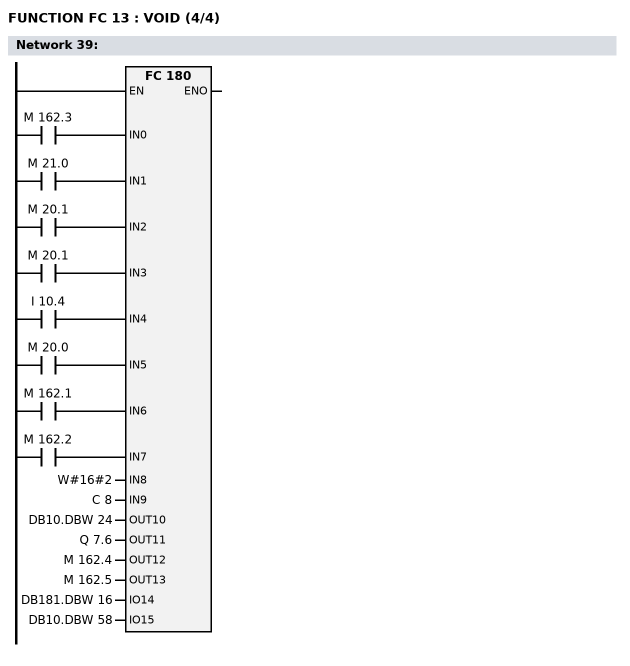

      A     M    162.3;
      =     L      4.0;
      BLD   103;
      A     M     21.0;
      =     L      4.1;
      BLD   103;
      A     M     20.1;
      =     L      4.2;
      BLD   103;
      A     M     20.1;
      =     L      4.3;
      BLD   103;
      A     I     10.4;
      =     L      4.4;
      BLD   103;
      A     M     20.0;
      =     L      4.5;
      BLD   103;
      A     M    162.1;
      =     L      4.6;
      BLD   103;
      A     M    162.2;
      =     L      4.7;
      BLD   103;
      CALL FC   180 (
           IN0                      := L      4.0,
           IN1                      := L      4.1,
           IN2                      := L      4.2,
           IN3                      := L      4.3,
           IN4                      := L      4.4,
           IN5                      := L      4.5,
           IN6                      := L      4.6,
           IN7                      := L      4.7,
           IN8                      := W#16#2,
           IN9                      := C      8,
           OUT10                    := DB10.DBW   24,
           OUT11                    := Q      7.6,
           OUT12                    := M    162.4,
           OUT13                    := M    162.5,
           IO14                     := DB181.DBW   16,
           IO15                     := DB10.DBW   58);
      NOP   0;
END_FUNCTION

FUNCTION FC 14 : VOID
TITLE =
AUTHOR : Xaadem <yalanci63@yahoo.com>
FAMILY : DRIVES
NAME : DRIVES
VERSION : 0.1


VAR_TEMP
  TEMP0 : REAL ;
END_VAR
BEGIN
NETWORK
TITLE =
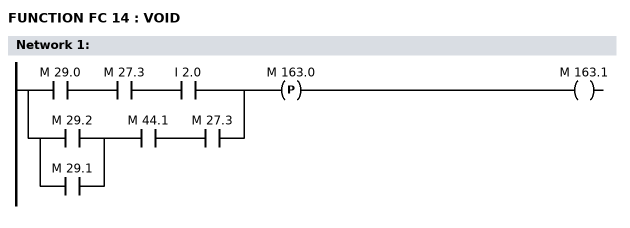

      A(    ;
      A     M     29.0;
      A     M     27.3;
      A     I      2.0;
      O     ;
      A(    ;
      O     M     29.2;
      O     M     29.1;
      )     ;
      A     M     44.1;
      A     M     27.3;
      )     ;
      FP    M    163.0;
      =     M    163.1;
NETWORK
TITLE =

      A     M     29.0;
      AN    I      2.1;
      O     ;
      A(    ;
      O     M     29.2;
      O     M     29.1;
      )     ;
      AN    M     44.1;
      A(    ;
      AN    T     25;
      L     DB2.DBW   58;
      SD    T     29;
      NOP   0;
      NOP   0;
      NOP   0;
      A     T     29;
      )     ;
      O     M     11.1;
      =     M    163.2;
NETWORK
TITLE =

      AN    M    179.0;
      AN    M    180.0;
      AN    M    181.0;
      AN    M    182.0;
      AN    M    183.0;
      A(    ;
      O     I      1.6;
      O     I      4.2;
      )     ;
      A(    ;
      A(    ;
      A     I     10.5;
      L     DB2.DBW   60;
      SD    T     30;
      NOP   0;
      NOP   0;
      NOP   0;
      A     T     30;
      )     ;
      AN    M    155.7;
      NOT   ;
      )     ;
      AN    M    206.0;
      AN    M    207.0;
      =     M    163.3;
NETWORK
TITLE =
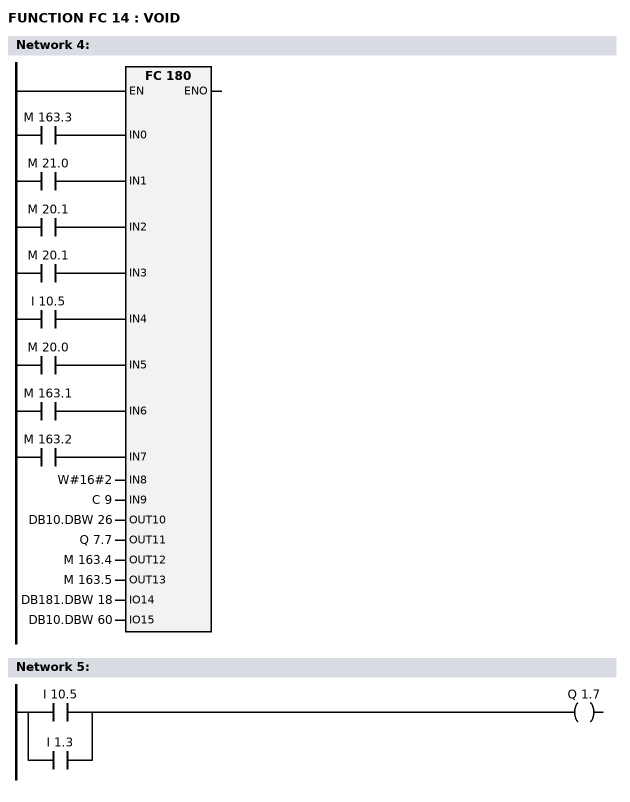

      A     M    163.3;
      =     L      4.0;
      BLD   103;
      A     M     21.0;
      =     L      4.1;
      BLD   103;
      A     M     20.1;
      =     L      4.2;
      BLD   103;
      A     M     20.1;
      =     L      4.3;
      BLD   103;
      A     I     10.5;
      =     L      4.4;
      BLD   103;
      A     M     20.0;
      =     L      4.5;
      BLD   103;
      A     M    163.1;
      =     L      4.6;
      BLD   103;
      A     M    163.2;
      =     L      4.7;
      BLD   103;
      CALL FC   180 (
           IN0                      := L      4.0,
           IN1                      := L      4.1,
           IN2                      := L      4.2,
           IN3                      := L      4.3,
           IN4                      := L      4.4,
           IN5                      := L      4.5,
           IN6                      := L      4.6,
           IN7                      := L      4.7,
           IN8                      := W#16#2,
           IN9                      := C      9,
           OUT10                    := DB10.DBW   26,
           OUT11                    := Q      7.7,
           OUT12                    := M    163.4,
           OUT13                    := M    163.5,
           IO14                     := DB181.DBW   18,
           IO15                     := DB10.DBW   60);
      NOP   0;
NETWORK
TITLE =

      O     I     10.5;
      O     I      1.3;
      =     Q      1.7;
END_FUNCTION

FUNCTION FC 15 : VOID
TITLE =
AUTHOR : Xaadem <yalanci63@yahoo.com>
FAMILY : DRIVES
NAME : DRIVES
VERSION : 0.1


VAR_TEMP
  TEMP0 : REAL ;
END_VAR
BEGIN
NETWORK
TITLE =

      A     I      0.2;
      AN    M    164.4;
      A(    ;
      A(    ;
      O     Q      0.0;
      O     I      1.0;
      O     I      2.0;
      O     I      2.4;
      O     I      2.6;
      O     I      2.7;
      O(    ;
      A     I      4.1;
      FP    M    209.2;
      )     ;
      )     ;
      =     M    209.3;
      A     M    209.3;
      )     ;
      FP    M    164.0;
      =     M    164.1;
NETWORK
TITLE =

      A(    ;
      A     M     38.0;
      A(    ;
      O     I     11.4;
      O     I     12.5;
      )     ;
      L     DB2.DBW   62;
      SD    T     31;
      NOP   0;
      NOP   0;
      NOP   0;
      A     T     31;
      )     ;
      FP    M    209.0;
      =     M    164.2;
NETWORK
TITLE =
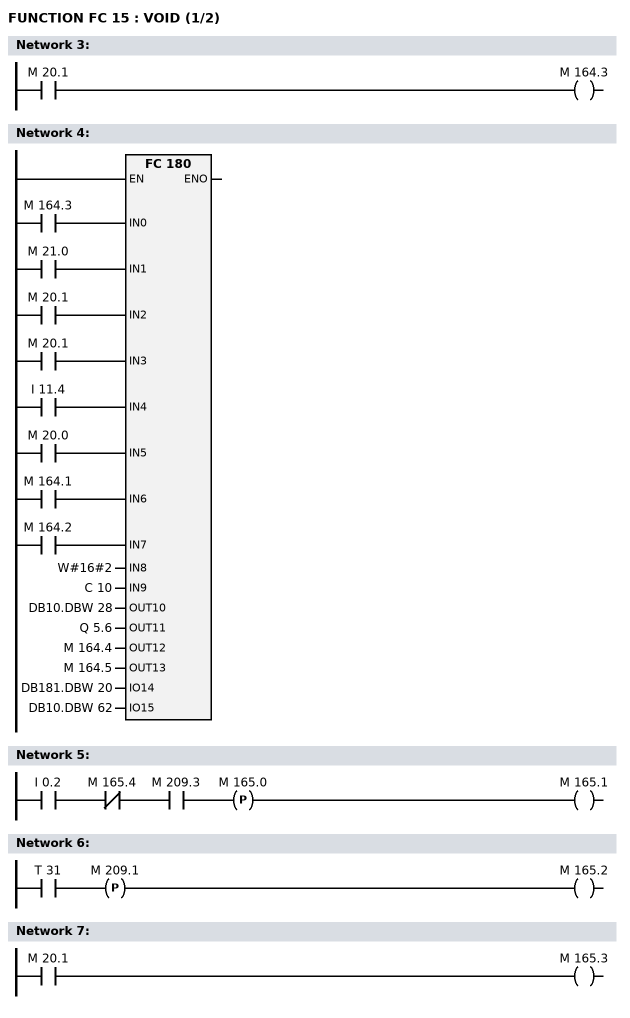

      A     M     20.1;
      =     M    164.3;
NETWORK
TITLE =

      A     M    164.3;
      =     L      4.0;
      BLD   103;
      A     M     21.0;
      =     L      4.1;
      BLD   103;
      A     M     20.1;
      =     L      4.2;
      BLD   103;
      A     M     20.1;
      =     L      4.3;
      BLD   103;
      A     I     11.4;
      =     L      4.4;
      BLD   103;
      A     M     20.0;
      =     L      4.5;
      BLD   103;
      A     M    164.1;
      =     L      4.6;
      BLD   103;
      A     M    164.2;
      =     L      4.7;
      BLD   103;
      CALL FC   180 (
           IN0                      := L      4.0,
           IN1                      := L      4.1,
           IN2                      := L      4.2,
           IN3                      := L      4.3,
           IN4                      := L      4.4,
           IN5                      := L      4.5,
           IN6                      := L      4.6,
           IN7                      := L      4.7,
           IN8                      := W#16#2,
           IN9                      := C     10,
           OUT10                    := DB10.DBW   28,
           OUT11                    := Q      5.6,
           OUT12                    := M    164.4,
           OUT13                    := M    164.5,
           IO14                     := DB181.DBW   20,
           IO15                     := DB10.DBW   62);
      NOP   0;
NETWORK
TITLE =

      A     I      0.2;
      AN    M    165.4;
      A     M    209.3;
      FP    M    165.0;
      =     M    165.1;
NETWORK
TITLE =

      A     T     31;
      FP    M    209.1;
      =     M    165.2;
NETWORK
TITLE =

      A     M     20.1;
      =     M    165.3;
NETWORK
TITLE =
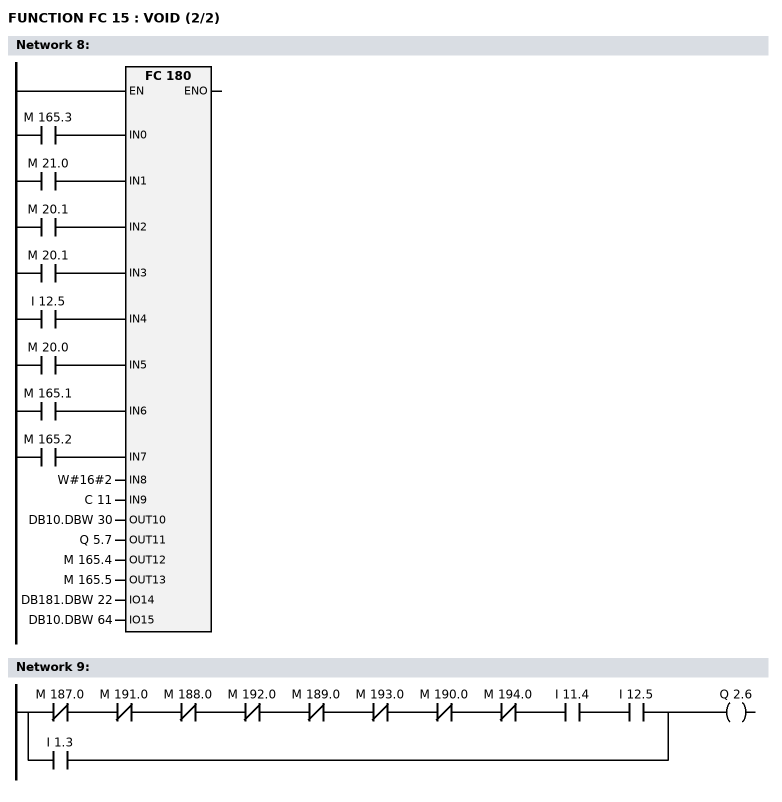

      A     M    165.3;
      =     L      4.0;
      BLD   103;
      A     M     21.0;
      =     L      4.1;
      BLD   103;
      A     M     20.1;
      =     L      4.2;
      BLD   103;
      A     M     20.1;
      =     L      4.3;
      BLD   103;
      A     I     12.5;
      =     L      4.4;
      BLD   103;
      A     M     20.0;
      =     L      4.5;
      BLD   103;
      A     M    165.1;
      =     L      4.6;
      BLD   103;
      A     M    165.2;
      =     L      4.7;
      BLD   103;
      CALL FC   180 (
           IN0                      := L      4.0,
           IN1                      := L      4.1,
           IN2                      := L      4.2,
           IN3                      := L      4.3,
           IN4                      := L      4.4,
           IN5                      := L      4.5,
           IN6                      := L      4.6,
           IN7                      := L      4.7,
           IN8                      := W#16#2,
           IN9                      := C     11,
           OUT10                    := DB10.DBW   30,
           OUT11                    := Q      5.7,
           OUT12                    := M    165.4,
           OUT13                    := M    165.5,
           IO14                     := DB181.DBW   22,
           IO15                     := DB10.DBW   64);
      NOP   0;
NETWORK
TITLE =

      AN    M    187.0;
      AN    M    191.0;
      AN    M    188.0;
      AN    M    192.0;
      AN    M    189.0;
      AN    M    193.0;
      AN    M    190.0;
      AN    M    194.0;
      A     I     11.4;
      A     I     12.5;
      O     I      1.3;
      =     Q      2.6;
END_FUNCTION

FUNCTION FC 20 : VOID
TITLE =
AUTHOR : Xaadem <yalanci63@yahoo.com>
FAMILY : ANALOGUE
NAME : ANALOGUE
VERSION : 0.1


VAR_TEMP
  TEMP0 : WORD ;
  TEMP1 : REAL ;
  TEMP2 : REAL ;
END_VAR
BEGIN
NETWORK
TITLE =

      L     ID   105;
      DTR   ;
      T     #TEMP2;
      NOP   0;
NETWORK
TITLE =

      L     ID   105;
      DTR   ;
      T     DB10.DBD  264;
      NOP   0;
NETWORK
TITLE =

      A(    ;
      A     I    108.0;
      FP    M    500.0;
      L     DB2.DBW  200;
      SF    T    100;
      NOP   0;
      NOP   0;
      NOP   0;
      A     T    100;
      )     ;
      NOT   ;
      A(    ;
      A(    ;
      O     I      5.5;
      O     I      6.4;
      )     ;
      L     DB2.DBW  210;
      SD    T    105;
      NOP   0;
      NOP   0;
      NOP   0;
      A     T    105;
      )     ;
      =     M    500.1;
NETWORK
TITLE =
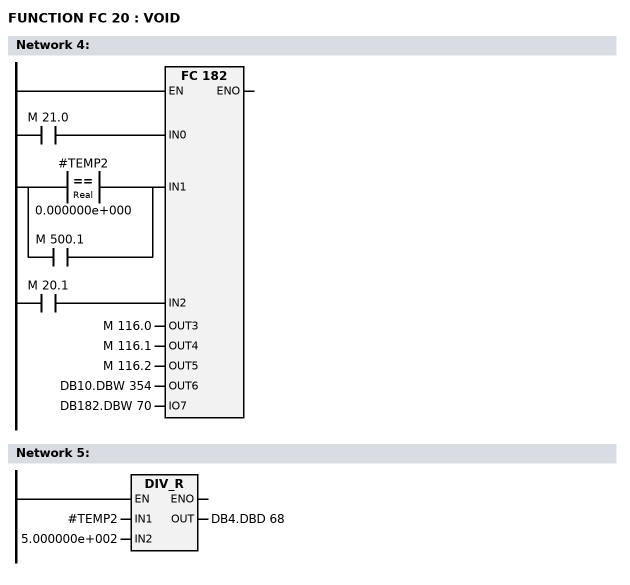

      A     M     21.0;
      =     L     10.0;
      BLD   103;
      A(    ;
      O(    ;
      L     #TEMP2;
      L     0.000000e+000;
      ==R   ;
      )     ;
      O     M    500.1;
      )     ;
      =     L     10.1;
      BLD   103;
      A     M     20.1;
      =     L     10.2;
      BLD   103;
      CALL FC   182 (
           IN0                      := L     10.0,
           IN1                      := L     10.1,
           IN2                      := L     10.2,
           OUT3                     := M    116.0,
           OUT4                     := M    116.1,
           OUT5                     := M    116.2,
           OUT6                     := DB10.DBW  354,
           IO7                      := DB182.DBW   70);
      NOP   0;
NETWORK
TITLE =

      L     #TEMP2;
      L     5.000000e+002;
      /R    ;
      T     DB4.DBD   68;
      NOP   0;
NETWORK
TITLE =

      A(    ;
      L     DB4.DBD   68;
      L     DB4.DBD   76;
      >=R   ;
      )     ;
      A(    ;
      L     DB4.DBD   68;
      L     DB4.DBD   72;
      <=R   ;
      )     ;
      =     L     10.0;
      A     L     10.0;
      BLD   102;
      =     M    172.0;
      O     L     10.0;
      O     I      1.3;
      =     Q      1.2;
      A     L     10.0;
      BLD   102;
      =     Q      3.7;
NETWORK
TITLE =

      A(    ;
      L     DB4.DBD   68;
      L     DB4.DBD   84;
      >=R   ;
      )     ;
      A(    ;
      L     DB4.DBD   68;
      L     DB4.DBD   80;
      <=R   ;
      )     ;
      =     L     10.0;
      A     L     10.0;
      BLD   102;
      =     M    172.1;
      O     L     10.0;
      O     I      1.3;
      =     Q      1.3;
      A     L     10.0;
      BLD   102;
      =     Q      4.0;
NETWORK
TITLE =
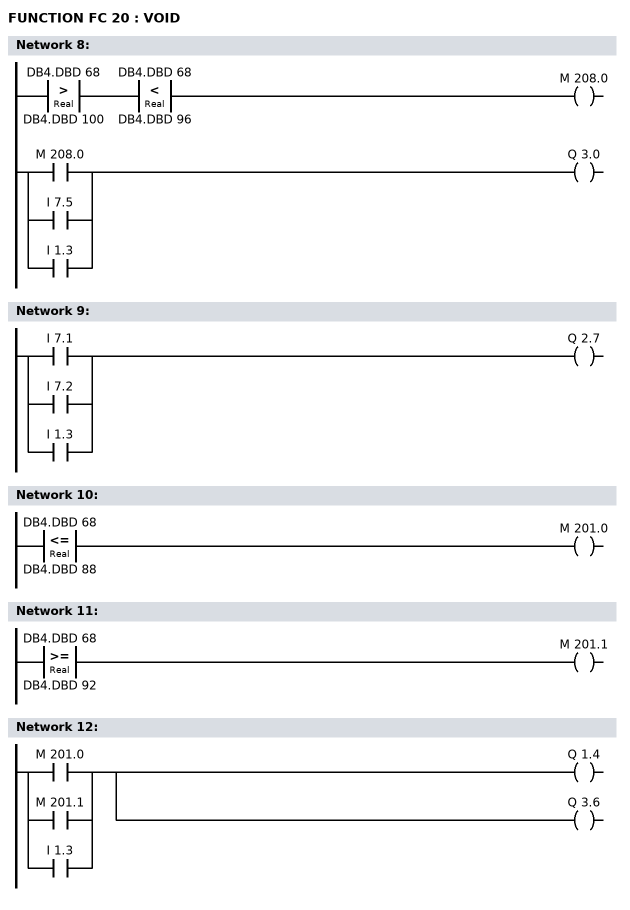

      A(    ;
      L     DB4.DBD   68;
      L     DB4.DBD  100;
      >R    ;
      )     ;
      A(    ;
      L     DB4.DBD   68;
      L     DB4.DBD   96;
      <R    ;
      )     ;
      =     M    208.0;
      A     M    208.0;
      O     I      7.5;
      O     I      1.3;
      =     Q      3.0;
NETWORK
TITLE =

      O     I      7.1;
      O     I      7.2;
      O     I      1.3;
      =     Q      2.7;
NETWORK
TITLE =

      L     DB4.DBD   68;
      L     DB4.DBD   88;
      <=R   ;
      =     M    201.0;
NETWORK
TITLE =

      L     DB4.DBD   68;
      L     DB4.DBD   92;
      >=R   ;
      =     M    201.1;
NETWORK
TITLE =

      O     M    201.0;
      O     M    201.1;
      O     I      1.3;
      =     Q      1.4;
      =     Q      3.6;
NETWORK
TITLE =

      A     M    200.6;
      A     M     20.1;
      =     L     10.0;
      A     L     10.0;
      JNB   M001;
      L     DW#16#80000000;
      T     QD   105;
M001: NOP   0;
      AN    L     10.0;
      JNB   M002;
      L     DW#16#0;
      T     QD   105;
M002: NOP   0;
NETWORK
TITLE =
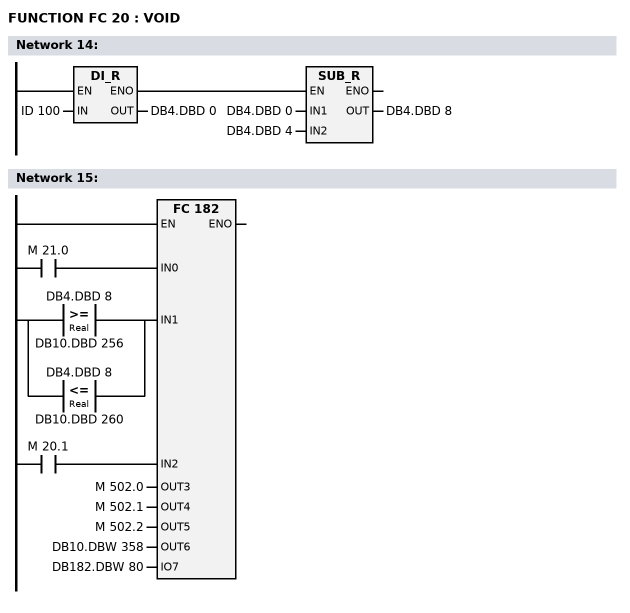

      A(    ;
      L     ID   100;
      DTR   ;
      T     DB4.DBD    0;
      SET   ;
      SAVE  ;
      CLR   ;
      A     BR;
      )     ;
      JNB   M003;
      L     DB4.DBD    0;
      L     DB4.DBD    4;
      -R    ;
      T     DB4.DBD    8;
M003: NOP   0;
NETWORK
TITLE =

      A     M     21.0;
      =     L     10.0;
      BLD   103;
      A(    ;
      O(    ;
      L     DB4.DBD    8;
      L     DB10.DBD  256;
      >=R   ;
      )     ;
      O(    ;
      L     DB4.DBD    8;
      L     DB10.DBD  260;
      <=R   ;
      )     ;
      )     ;
      =     L     10.1;
      BLD   103;
      A     M     20.1;
      =     L     10.2;
      BLD   103;
      CALL FC   182 (
           IN0                      := L     10.0,
           IN1                      := L     10.1,
           IN2                      := L     10.2,
           OUT3                     := M    502.0,
           OUT4                     := M    502.1,
           OUT5                     := M    502.2,
           OUT6                     := DB10.DBW  358,
           IO7                      := DB182.DBW   80);
      NOP   0;
NETWORK
TITLE =

      A(    ;
      L     DB4.DBD    8;
      L     DB10.DBD  248;
      >=R   ;
      )     ;
      =     M    503.1;
      A     M    503.1;
      O(    ;
      A(    ;
      L     DB4.DBD    8;
      L     DB10.DBD  252;
      <=R   ;
      )     ;
      =     M    503.2;
      A     M    503.2;
      )     ;
      =     M    503.0;
NETWORK
TITLE =

      A(    ;
      A     I    103.0;
      FP    M    501.0;
      L     DB2.DBW  202;
      SF    T    101;
      NOP   0;
      NOP   0;
      NOP   0;
      A     T    101;
      )     ;
      NOT   ;
      A     T    105;
      =     M    501.1;
NETWORK
TITLE =
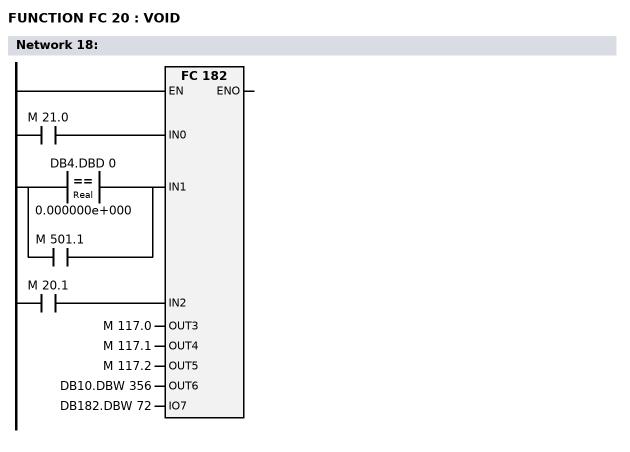

      A     M     21.0;
      =     L     10.0;
      BLD   103;
      A(    ;
      O(    ;
      L     DB4.DBD    0;
      L     0.000000e+000;
      ==R   ;
      )     ;
      O     M    501.1;
      )     ;
      =     L     10.1;
      BLD   103;
      A     M     20.1;
      =     L     10.2;
      BLD   103;
      CALL FC   182 (
           IN0                      := L     10.0,
           IN1                      := L     10.1,
           IN2                      := L     10.2,
           OUT3                     := M    117.0,
           OUT4                     := M    117.1,
           OUT5                     := M    117.2,
           OUT6                     := DB10.DBW  356,
           IO7                      := DB182.DBW   72);
      NOP   0;
NETWORK
TITLE =

      A     M     20.1;
      A     M    200.5;
      =     L     10.0;
      A     L     10.0;
      JNB   M004;
      L     DW#16#80000000;
      T     QD   100;
M004: NOP   0;
      AN    L     10.0;
      JNB   M005;
      L     DW#16#0;
      T     QD   100;
M005: NOP   0;
NETWORK
TITLE =
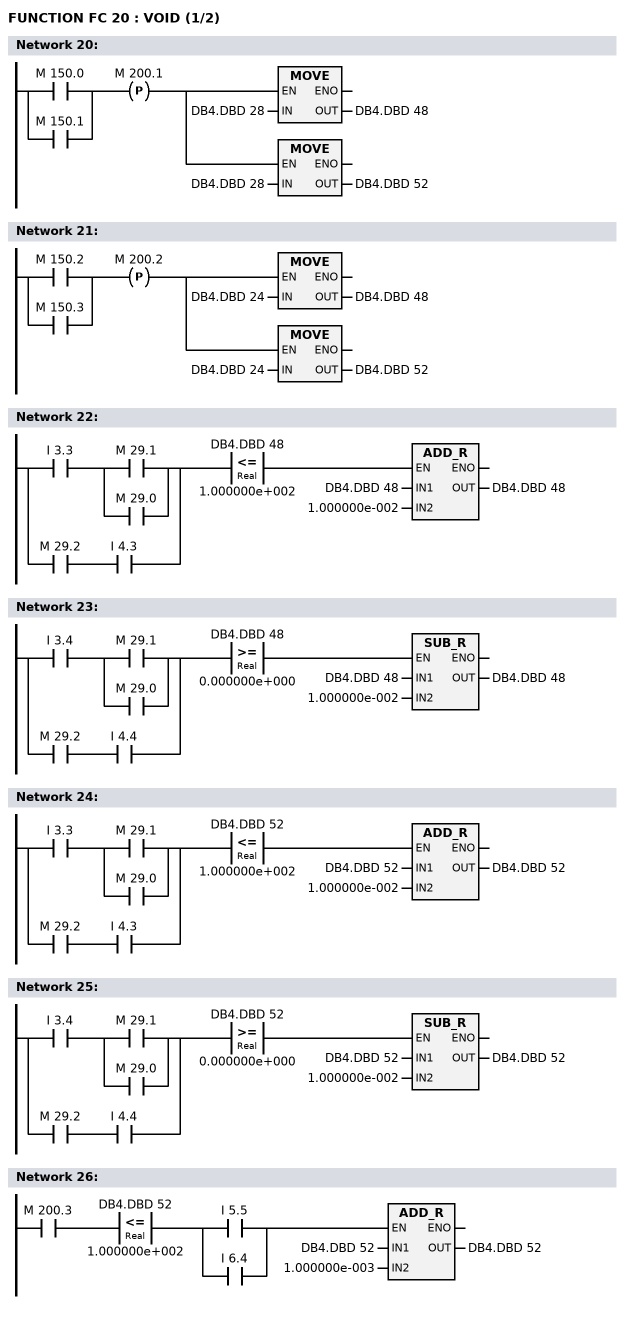

      A(    ;
      O     M    150.0;
      O     M    150.1;
      )     ;
      FP    M    200.1;
      =     L     10.0;
      A     L     10.0;
      JNB   M006;
      L     DB4.DBD   28;
      T     DB4.DBD   48;
M006: NOP   0;
      A     L     10.0;
      JNB   M007;
      L     DB4.DBD   28;
      T     DB4.DBD   52;
M007: NOP   0;
NETWORK
TITLE =

      A(    ;
      O     M    150.2;
      O     M    150.3;
      )     ;
      FP    M    200.2;
      =     L     10.0;
      A     L     10.0;
      JNB   M008;
      L     DB4.DBD   24;
      T     DB4.DBD   48;
M008: NOP   0;
      A     L     10.0;
      JNB   M009;
      L     DB4.DBD   24;
      T     DB4.DBD   52;
M009: NOP   0;
NETWORK
TITLE =

      A(    ;
      A     I      3.3;
      A(    ;
      O     M     29.1;
      O     M     29.0;
      )     ;
      O     ;
      A     M     29.2;
      A     I      4.3;
      )     ;
      A(    ;
      L     DB4.DBD   48;
      L     1.000000e+002;
      <=R   ;
      )     ;
      JNB   M00a;
      L     DB4.DBD   48;
      L     1.000000e-002;
      +R    ;
      T     DB4.DBD   48;
M00a: NOP   0;
NETWORK
TITLE =

      A(    ;
      A     I      3.4;
      A(    ;
      O     M     29.1;
      O     M     29.0;
      )     ;
      O     ;
      A     M     29.2;
      A     I      4.4;
      )     ;
      A(    ;
      L     DB4.DBD   48;
      L     0.000000e+000;
      >=R   ;
      )     ;
      JNB   M00b;
      L     DB4.DBD   48;
      L     1.000000e-002;
      -R    ;
      T     DB4.DBD   48;
M00b: NOP   0;
NETWORK
TITLE =

      A(    ;
      A     I      3.3;
      A(    ;
      O     M     29.1;
      O     M     29.0;
      )     ;
      O     ;
      A     M     29.2;
      A     I      4.3;
      )     ;
      A(    ;
      L     DB4.DBD   52;
      L     1.000000e+002;
      <=R   ;
      )     ;
      JNB   M00c;
      L     DB4.DBD   52;
      L     1.000000e-002;
      +R    ;
      T     DB4.DBD   52;
M00c: NOP   0;
NETWORK
TITLE =

      A(    ;
      A     I      3.4;
      A(    ;
      O     M     29.1;
      O     M     29.0;
      )     ;
      O     ;
      A     M     29.2;
      A     I      4.4;
      )     ;
      A(    ;
      L     DB4.DBD   52;
      L     0.000000e+000;
      >=R   ;
      )     ;
      JNB   M00d;
      L     DB4.DBD   52;
      L     1.000000e-002;
      -R    ;
      T     DB4.DBD   52;
M00d: NOP   0;
NETWORK
TITLE =

      A     M    200.3;
      A(    ;
      L     DB4.DBD   52;
      L     1.000000e+002;
      <=R   ;
      )     ;
      A(    ;
      O     I      5.5;
      O     I      6.4;
      )     ;
      JNB   M00e;
      L     DB4.DBD   52;
      L     1.000000e-003;
      +R    ;
      T     DB4.DBD   52;
M00e: NOP   0;
NETWORK
TITLE =
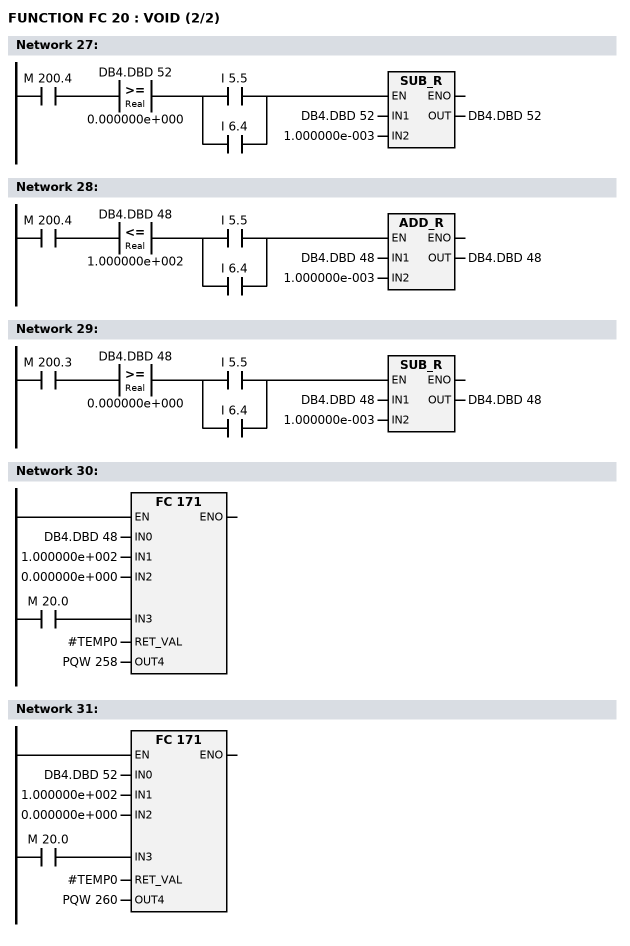

      A     M    200.4;
      A(    ;
      L     DB4.DBD   52;
      L     0.000000e+000;
      >=R   ;
      )     ;
      A(    ;
      O     I      5.5;
      O     I      6.4;
      )     ;
      JNB   M00f;
      L     DB4.DBD   52;
      L     1.000000e-003;
      -R    ;
      T     DB4.DBD   52;
M00f: NOP   0;
NETWORK
TITLE =

      A     M    200.4;
      A(    ;
      L     DB4.DBD   48;
      L     1.000000e+002;
      <=R   ;
      )     ;
      A(    ;
      O     I      5.5;
      O     I      6.4;
      )     ;
      JNB   M010;
      L     DB4.DBD   48;
      L     1.000000e-003;
      +R    ;
      T     DB4.DBD   48;
M010: NOP   0;
NETWORK
TITLE =

      A     M    200.3;
      A(    ;
      L     DB4.DBD   48;
      L     0.000000e+000;
      >=R   ;
      )     ;
      A(    ;
      O     I      5.5;
      O     I      6.4;
      )     ;
      JNB   M011;
      L     DB4.DBD   48;
      L     1.000000e-003;
      -R    ;
      T     DB4.DBD   48;
M011: NOP   0;
NETWORK
TITLE =

      A     M     20.0;
      =     L     10.0;
      BLD   103;
      CALL FC   171 (
           IN0                      := DB4.DBD   48,
           IN1                      := 1.000000e+002,
           IN2                      := 0.000000e+000,
           IN3                      := L     10.0,
           RET_VAL                  := #TEMP0,
           OUT4                     := PQW  258);
      NOP   0;
NETWORK
TITLE =

      A     M     20.0;
      =     L     10.0;
      BLD   103;
      CALL FC   171 (
           IN0                      := DB4.DBD   52,
           IN1                      := 1.000000e+002,
           IN2                      := 0.000000e+000,
           IN3                      := L     10.0,
           RET_VAL                  := #TEMP0,
           OUT4                     := PQW  260);
      NOP   0;
NETWORK
TITLE =

      A     I      5.5;
      A     I      6.4;
      =     L     10.0;
      A     L     10.0;
      JNB   M012;
      L     DB4.DBD   48;
      T     DB4.DBD   20;
M012: NOP   0;
      AN    L     10.0;
      JNB   M013;
      L     0.000000e+000;
      T     DB4.DBD   20;
M013: NOP   0;
NETWORK
TITLE =
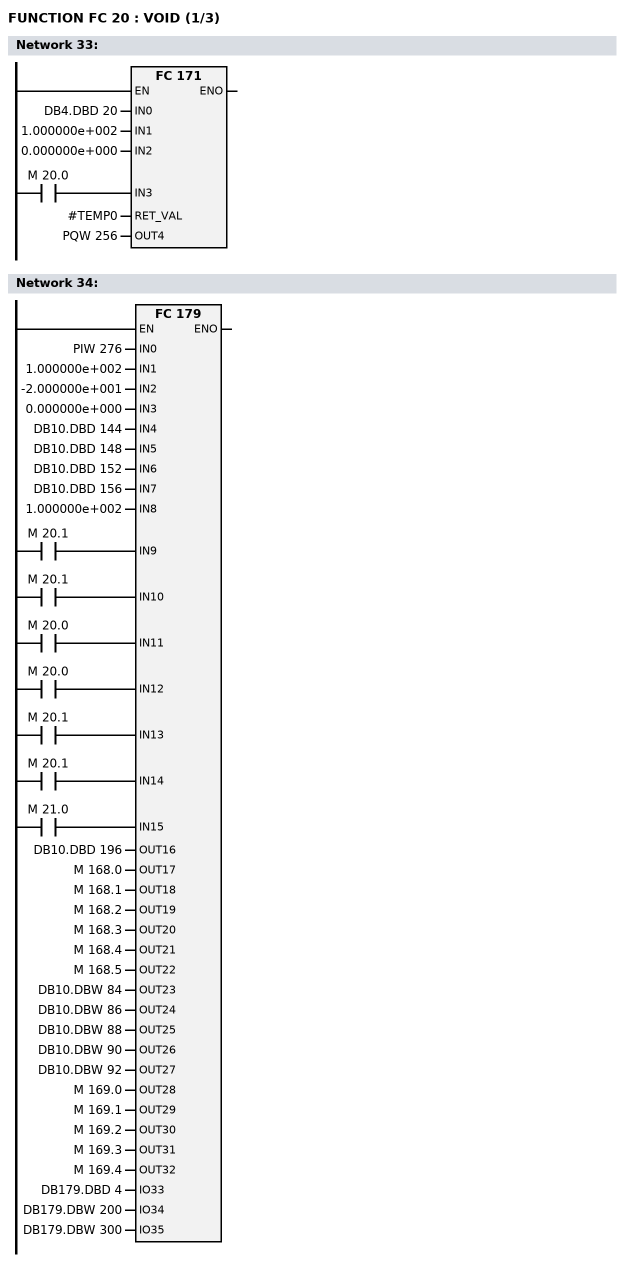

      A     M     20.0;
      =     L     10.0;
      BLD   103;
      CALL FC   171 (
           IN0                      := DB4.DBD   20,
           IN1                      := 1.000000e+002,
           IN2                      := 0.000000e+000,
           IN3                      := L     10.0,
           RET_VAL                  := #TEMP0,
           OUT4                     := PQW  256);
      NOP   0;
NETWORK
TITLE =

      A     M     20.1;
      =     L     10.0;
      BLD   103;
      A     M     20.1;
      =     L     10.1;
      BLD   103;
      A     M     20.0;
      =     L     10.2;
      BLD   103;
      A     M     20.0;
      =     L     10.3;
      BLD   103;
      A     M     20.1;
      =     L     10.4;
      BLD   103;
      A     M     20.1;
      =     L     10.5;
      BLD   103;
      A     M     21.0;
      =     L     10.6;
      BLD   103;
      CALL FC   179 (
           IN0                      := PIW  276,
           IN1                      := 1.000000e+002,
           IN2                      := -2.000000e+001,
           IN3                      := 0.000000e+000,
           IN4                      := DB10.DBD  144,
           IN5                      := DB10.DBD  148,
           IN6                      := DB10.DBD  152,
           IN7                      := DB10.DBD  156,
           IN8                      := 1.000000e+002,
           IN9                      := L     10.0,
           IN10                     := L     10.1,
           IN11                     := L     10.2,
           IN12                     := L     10.3,
           IN13                     := L     10.4,
           IN14                     := L     10.5,
           IN15                     := L     10.6,
           OUT16                    := DB10.DBD  196,
           OUT17                    := M    168.0,
           OUT18                    := M    168.1,
           OUT19                    := M    168.2,
           OUT20                    := M    168.3,
           OUT21                    := M    168.4,
           OUT22                    := M    168.5,
           OUT23                    := DB10.DBW   84,
           OUT24                    := DB10.DBW   86,
           OUT25                    := DB10.DBW   88,
           OUT26                    := DB10.DBW   90,
           OUT27                    := DB10.DBW   92,
           OUT28                    := M    169.0,
           OUT29                    := M    169.1,
           OUT30                    := M    169.2,
           OUT31                    := M    169.3,
           OUT32                    := M    169.4,
           IO33                     := DB179.DBD    4,
           IO34                     := DB179.DBW  200,
           IO35                     := DB179.DBW  300);
      NOP   0;
NETWORK
TITLE =
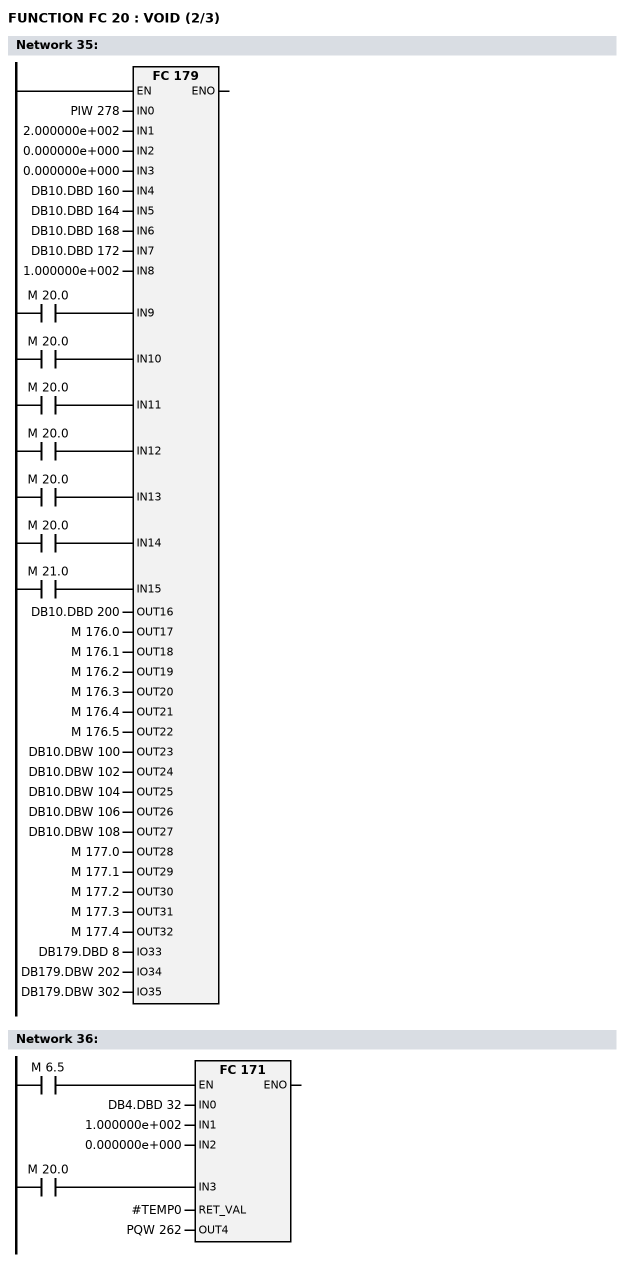

      A     M     20.0;
      =     L     10.0;
      BLD   103;
      A     M     20.0;
      =     L     10.1;
      BLD   103;
      A     M     20.0;
      =     L     10.2;
      BLD   103;
      A     M     20.0;
      =     L     10.3;
      BLD   103;
      A     M     20.0;
      =     L     10.4;
      BLD   103;
      A     M     20.0;
      =     L     10.5;
      BLD   103;
      A     M     21.0;
      =     L     10.6;
      BLD   103;
      CALL FC   179 (
           IN0                      := PIW  278,
           IN1                      := 2.000000e+002,
           IN2                      := 0.000000e+000,
           IN3                      := 0.000000e+000,
           IN4                      := DB10.DBD  160,
           IN5                      := DB10.DBD  164,
           IN6                      := DB10.DBD  168,
           IN7                      := DB10.DBD  172,
           IN8                      := 1.000000e+002,
           IN9                      := L     10.0,
           IN10                     := L     10.1,
           IN11                     := L     10.2,
           IN12                     := L     10.3,
           IN13                     := L     10.4,
           IN14                     := L     10.5,
           IN15                     := L     10.6,
           OUT16                    := DB10.DBD  200,
           OUT17                    := M    176.0,
           OUT18                    := M    176.1,
           OUT19                    := M    176.2,
           OUT20                    := M    176.3,
           OUT21                    := M    176.4,
           OUT22                    := M    176.5,
           OUT23                    := DB10.DBW  100,
           OUT24                    := DB10.DBW  102,
           OUT25                    := DB10.DBW  104,
           OUT26                    := DB10.DBW  106,
           OUT27                    := DB10.DBW  108,
           OUT28                    := M    177.0,
           OUT29                    := M    177.1,
           OUT30                    := M    177.2,
           OUT31                    := M    177.3,
           OUT32                    := M    177.4,
           IO33                     := DB179.DBD    8,
           IO34                     := DB179.DBW  202,
           IO35                     := DB179.DBW  302);
      NOP   0;
NETWORK
TITLE =

      A     M     20.0;
      =     L     10.0;
      BLD   103;
      A     M      6.5;
      JNB   M014;
      CALL FC   171 (
           IN0                      := DB4.DBD   32,
           IN1                      := 1.000000e+002,
           IN2                      := 0.000000e+000,
           IN3                      := L     10.0,
           RET_VAL                  := #TEMP0,
           OUT4                     := PQW  262);
M014: NOP   0;
NETWORK
TITLE =
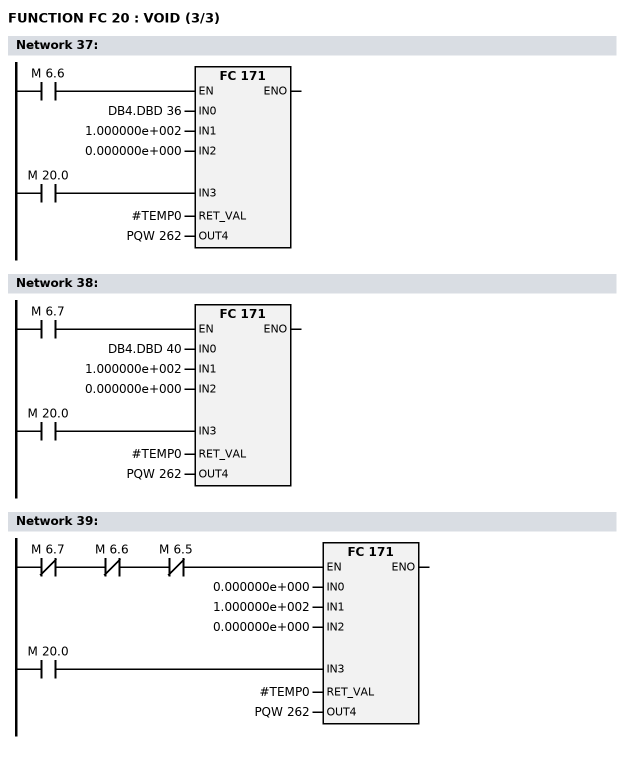

      A     M     20.0;
      =     L     10.0;
      BLD   103;
      A     M      6.6;
      JNB   M015;
      CALL FC   171 (
           IN0                      := DB4.DBD   36,
           IN1                      := 1.000000e+002,
           IN2                      := 0.000000e+000,
           IN3                      := L     10.0,
           RET_VAL                  := #TEMP0,
           OUT4                     := PQW  262);
M015: NOP   0;
NETWORK
TITLE =

      A     M     20.0;
      =     L     10.0;
      BLD   103;
      A     M      6.7;
      JNB   M016;
      CALL FC   171 (
           IN0                      := DB4.DBD   40,
           IN1                      := 1.000000e+002,
           IN2                      := 0.000000e+000,
           IN3                      := L     10.0,
           RET_VAL                  := #TEMP0,
           OUT4                     := PQW  262);
M016: NOP   0;
NETWORK
TITLE =

      A     M     20.0;
      =     L     10.0;
      BLD   103;
      AN    M      6.7;
      AN    M      6.6;
      AN    M      6.5;
      JNB   M017;
      CALL FC   171 (
           IN0                      := 0.000000e+000,
           IN1                      := 1.000000e+002,
           IN2                      := 0.000000e+000,
           IN3                      := L     10.0,
           RET_VAL                  := #TEMP0,
           OUT4                     := PQW  262);
M017: NOP   0;
END_FUNCTION

FUNCTION FC 21 : VOID
TITLE =
AUTHOR : Xaadem <yalanci63@yahoo.com>
FAMILY : DIGITAL
NAME : DIGITAL
VERSION : 0.1


VAR_TEMP
  TEMP0 : WORD ;
END_VAR
BEGIN
NETWORK
TITLE =

      A     M     21.0;
      =     L      2.0;
      BLD   103;
      AN    I      8.2;
      =     L      2.1;
      BLD   103;
      A(    ;
      AN    I      8.2;
      L     DB2.DBW   32;
      SD    T     16;
      NOP   0;
      NOP   0;
      NOP   0;
      A     T     16;
      )     ;
      =     L      2.2;
      BLD   103;
      CALL FC   182 (
           IN0                      := L      2.0,
           IN1                      := L      2.1,
           IN2                      := L      2.2,
           OUT3                     := M    155.0,
           OUT4                     := M    155.1,
           OUT5                     := M    155.2,
           OUT6                     := DB10.DBW   76,
           IO7                      := DB182.DBW    2);
      NOP   0;
NETWORK
TITLE =
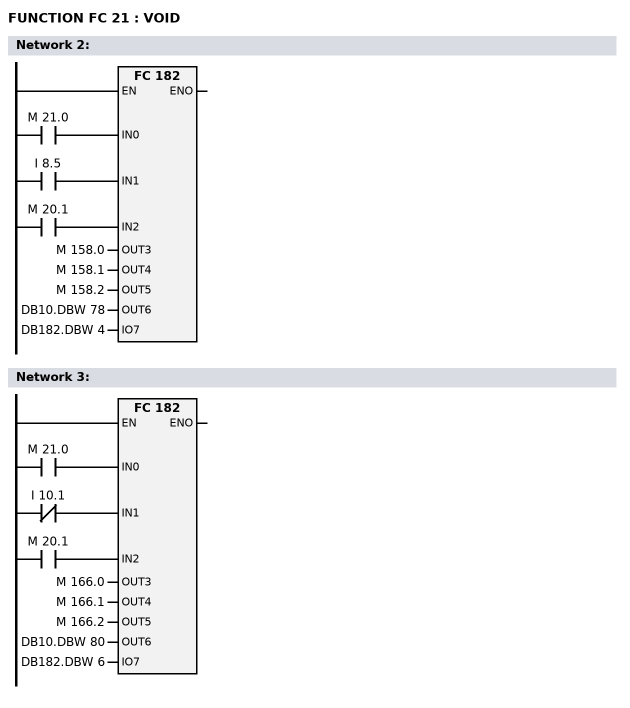

      A     M     21.0;
      =     L      2.0;
      BLD   103;
      A     I      8.5;
      =     L      2.1;
      BLD   103;
      A     M     20.1;
      =     L      2.2;
      BLD   103;
      CALL FC   182 (
           IN0                      := L      2.0,
           IN1                      := L      2.1,
           IN2                      := L      2.2,
           OUT3                     := M    158.0,
           OUT4                     := M    158.1,
           OUT5                     := M    158.2,
           OUT6                     := DB10.DBW   78,
           IO7                      := DB182.DBW    4);
      NOP   0;
NETWORK
TITLE =

      A     M     21.0;
      =     L      2.0;
      BLD   103;
      AN    I     10.1;
      =     L      2.1;
      BLD   103;
      A     M     20.1;
      =     L      2.2;
      BLD   103;
      CALL FC   182 (
           IN0                      := L      2.0,
           IN1                      := L      2.1,
           IN2                      := L      2.2,
           OUT3                     := M    166.0,
           OUT4                     := M    166.1,
           OUT5                     := M    166.2,
           OUT6                     := DB10.DBW   80,
           IO7                      := DB182.DBW    6);
      NOP   0;
NETWORK
TITLE =

      A     M     21.0;
      =     L      2.0;
      BLD   103;
      AN    I     10.2;
      =     L      2.1;
      BLD   103;
      A(    ;
      A     I      8.4;
      L     DB2.DBW   64;
      SD    T     32;
      NOP   0;
      NOP   0;
      NOP   0;
      A     T     32;
      )     ;
      =     L      2.2;
      BLD   103;
      CALL FC   182 (
           IN0                      := L      2.0,
           IN1                      := L      2.1,
           IN2                      := L      2.2,
           OUT3                     := M    167.0,
           OUT4                     := M    167.1,
           OUT5                     := M    167.2,
           OUT6                     := DB10.DBW   82,
           IO7                      := DB182.DBW    8);
      NOP   0;
NETWORK
TITLE =
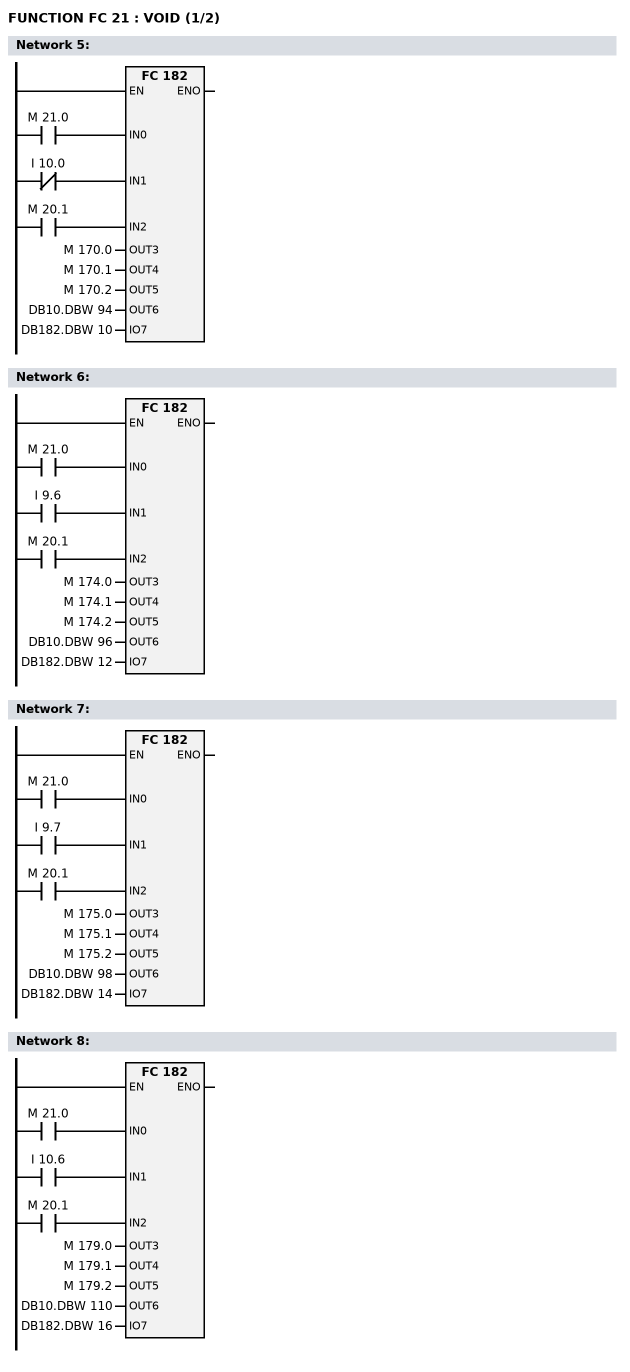

      A     M     21.0;
      =     L      2.0;
      BLD   103;
      AN    I     10.0;
      =     L      2.1;
      BLD   103;
      A     M     20.1;
      =     L      2.2;
      BLD   103;
      CALL FC   182 (
           IN0                      := L      2.0,
           IN1                      := L      2.1,
           IN2                      := L      2.2,
           OUT3                     := M    170.0,
           OUT4                     := M    170.1,
           OUT5                     := M    170.2,
           OUT6                     := DB10.DBW   94,
           IO7                      := DB182.DBW   10);
      NOP   0;
NETWORK
TITLE =

      A     M     21.0;
      =     L      2.0;
      BLD   103;
      A     I      9.6;
      =     L      2.1;
      BLD   103;
      A     M     20.1;
      =     L      2.2;
      BLD   103;
      CALL FC   182 (
           IN0                      := L      2.0,
           IN1                      := L      2.1,
           IN2                      := L      2.2,
           OUT3                     := M    174.0,
           OUT4                     := M    174.1,
           OUT5                     := M    174.2,
           OUT6                     := DB10.DBW   96,
           IO7                      := DB182.DBW   12);
      NOP   0;
NETWORK
TITLE =

      A     M     21.0;
      =     L      2.0;
      BLD   103;
      A     I      9.7;
      =     L      2.1;
      BLD   103;
      A     M     20.1;
      =     L      2.2;
      BLD   103;
      CALL FC   182 (
           IN0                      := L      2.0,
           IN1                      := L      2.1,
           IN2                      := L      2.2,
           OUT3                     := M    175.0,
           OUT4                     := M    175.1,
           OUT5                     := M    175.2,
           OUT6                     := DB10.DBW   98,
           IO7                      := DB182.DBW   14);
      NOP   0;
NETWORK
TITLE =

      A     M     21.0;
      =     L      2.0;
      BLD   103;
      A     I     10.6;
      =     L      2.1;
      BLD   103;
      A     M     20.1;
      =     L      2.2;
      BLD   103;
      CALL FC   182 (
           IN0                      := L      2.0,
           IN1                      := L      2.1,
           IN2                      := L      2.2,
           OUT3                     := M    179.0,
           OUT4                     := M    179.1,
           OUT5                     := M    179.2,
           OUT6                     := DB10.DBW  110,
           IO7                      := DB182.DBW   16);
      NOP   0;
NETWORK
TITLE =
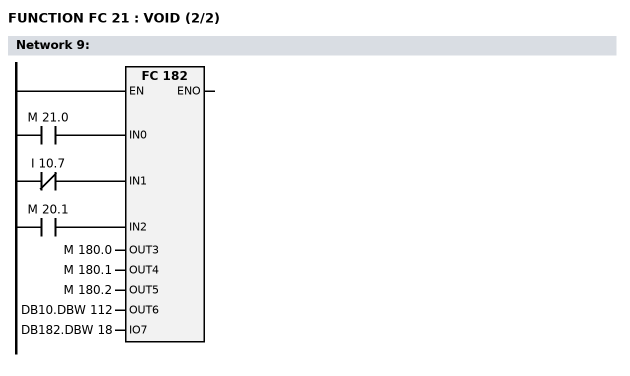

      A     M     21.0;
      =     L      2.0;
      BLD   103;
      AN    I     10.7;
      =     L      2.1;
      BLD   103;
      A     M     20.1;
      =     L      2.2;
      BLD   103;
      CALL FC   182 (
           IN0                      := L      2.0,
           IN1                      := L      2.1,
           IN2                      := L      2.2,
           OUT3                     := M    180.0,
           OUT4                     := M    180.1,
           OUT5                     := M    180.2,
           OUT6                     := DB10.DBW  112,
           IO7                      := DB182.DBW   18);
      NOP   0;
NETWORK
TITLE =

      A     M     21.0;
      =     L      2.0;
      BLD   103;
      A(    ;
      A     I     11.0;
      FP    M    184.0;
      L     DB2.DBW   38;
      SF    T     19;
      NOP   0;
      NOP   0;
      NOP   0;
      A     T     19;
      )     ;
      NOT   ;
      =     L      2.1;
      BLD   103;
      A(    ;
      A     I     10.5;
      L     DB2.DBW   36;
      SD    T     18;
      NOP   0;
      NOP   0;
      NOP   0;
      A     T     18;
      )     ;
      =     L      2.2;
      BLD   103;
      CALL FC   182 (
           IN0                      := L      2.0,
           IN1                      := L      2.1,
           IN2                      := L      2.2,
           OUT3                     := M    181.0,
           OUT4                     := M    181.1,
           OUT5                     := M    181.2,
           OUT6                     := DB10.DBW  310,
           IO7                      := DB182.DBW   20);
      NOP   0;
NETWORK
TITLE =

      A     M     21.0;
      =     L      2.0;
      BLD   103;
      A(    ;
      A     I     11.1;
      FP    M    184.1;
      L     DB2.DBW   40;
      SF    T     20;
      NOP   0;
      NOP   0;
      NOP   0;
      A     T     20;
      )     ;
      NOT   ;
      =     L      2.1;
      BLD   103;
      A     T     18;
      =     L      2.2;
      BLD   103;
      CALL FC   182 (
           IN0                      := L      2.0,
           IN1                      := L      2.1,
           IN2                      := L      2.2,
           OUT3                     := M    182.0,
           OUT4                     := M    182.1,
           OUT5                     := M    182.2,
           OUT6                     := DB10.DBW  312,
           IO7                      := DB182.DBW   22);
      NOP   0;
NETWORK
TITLE =
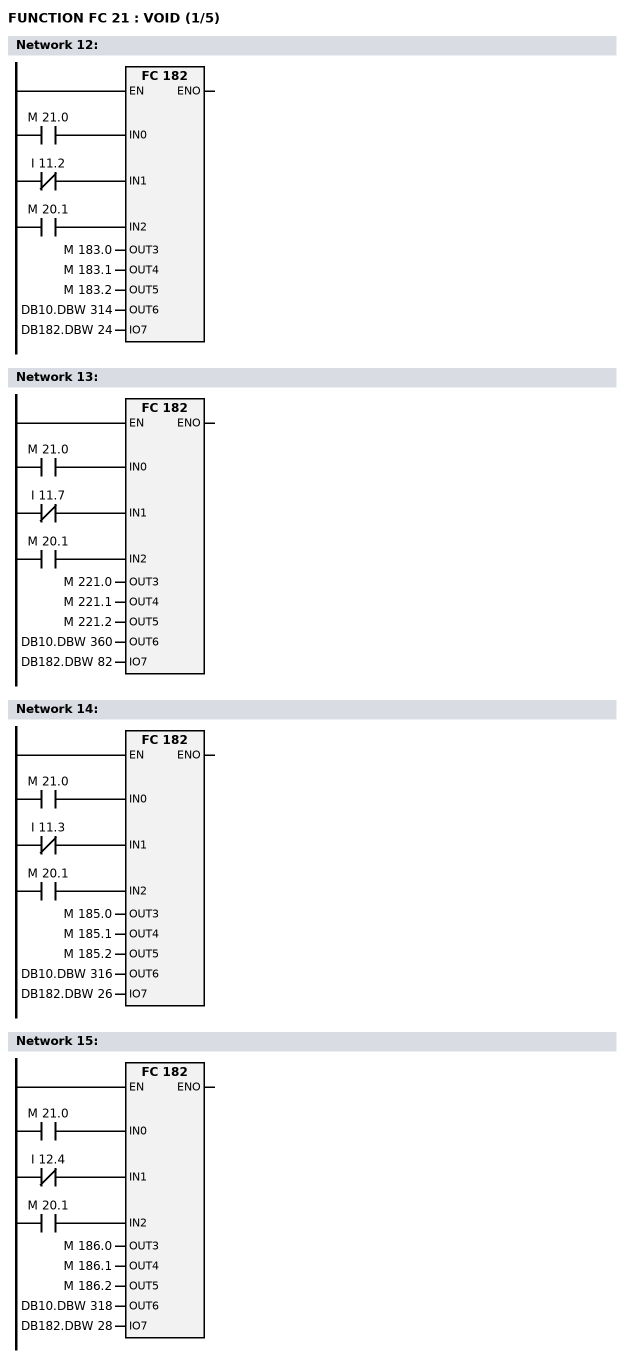

      A     M     21.0;
      =     L      2.0;
      BLD   103;
      AN    I     11.2;
      =     L      2.1;
      BLD   103;
      A     M     20.1;
      =     L      2.2;
      BLD   103;
      CALL FC   182 (
           IN0                      := L      2.0,
           IN1                      := L      2.1,
           IN2                      := L      2.2,
           OUT3                     := M    183.0,
           OUT4                     := M    183.1,
           OUT5                     := M    183.2,
           OUT6                     := DB10.DBW  314,
           IO7                      := DB182.DBW   24);
      NOP   0;
NETWORK
TITLE =

      A     M     21.0;
      =     L      2.0;
      BLD   103;
      AN    I     11.7;
      =     L      2.1;
      BLD   103;
      A     M     20.1;
      =     L      2.2;
      BLD   103;
      CALL FC   182 (
           IN0                      := L      2.0,
           IN1                      := L      2.1,
           IN2                      := L      2.2,
           OUT3                     := M    221.0,
           OUT4                     := M    221.1,
           OUT5                     := M    221.2,
           OUT6                     := DB10.DBW  360,
           IO7                      := DB182.DBW   82);
      NOP   0;
NETWORK
TITLE =

      A     M     21.0;
      =     L      2.0;
      BLD   103;
      AN    I     11.3;
      =     L      2.1;
      BLD   103;
      A     M     20.1;
      =     L      2.2;
      BLD   103;
      CALL FC   182 (
           IN0                      := L      2.0,
           IN1                      := L      2.1,
           IN2                      := L      2.2,
           OUT3                     := M    185.0,
           OUT4                     := M    185.1,
           OUT5                     := M    185.2,
           OUT6                     := DB10.DBW  316,
           IO7                      := DB182.DBW   26);
      NOP   0;
NETWORK
TITLE =

      A     M     21.0;
      =     L      2.0;
      BLD   103;
      AN    I     12.4;
      =     L      2.1;
      BLD   103;
      A     M     20.1;
      =     L      2.2;
      BLD   103;
      CALL FC   182 (
           IN0                      := L      2.0,
           IN1                      := L      2.1,
           IN2                      := L      2.2,
           OUT3                     := M    186.0,
           OUT4                     := M    186.1,
           OUT5                     := M    186.2,
           OUT6                     := DB10.DBW  318,
           IO7                      := DB182.DBW   28);
      NOP   0;
NETWORK
TITLE =
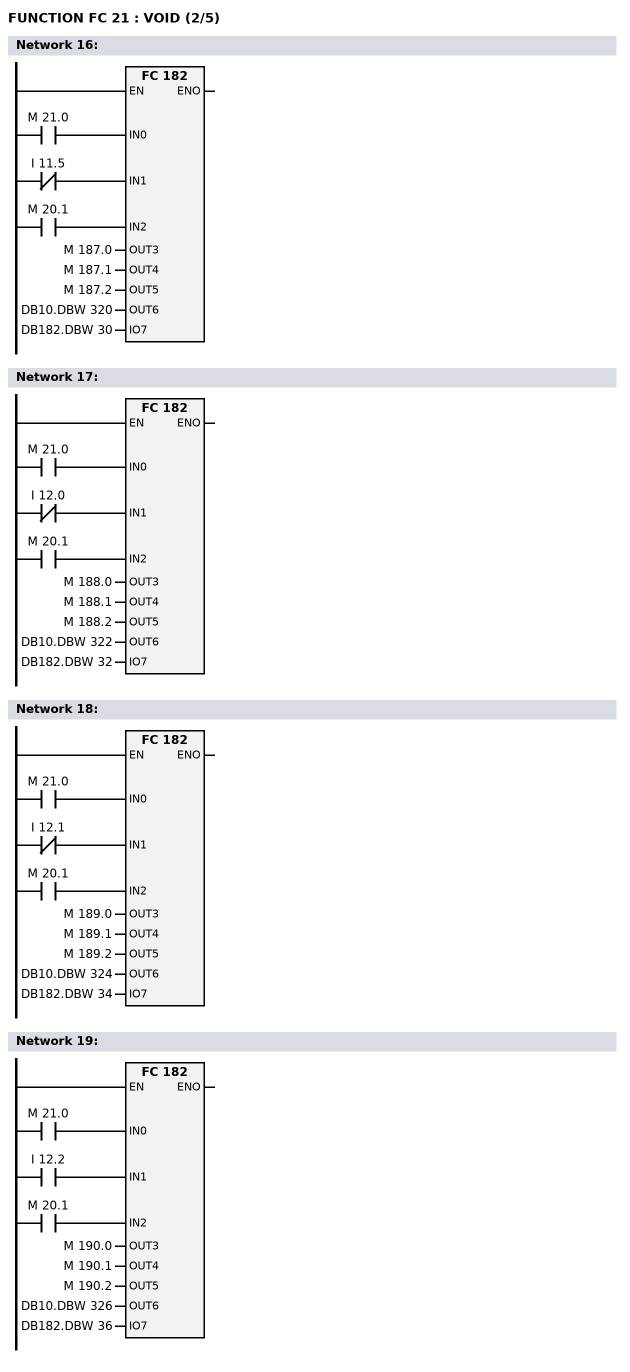

      A     M     21.0;
      =     L      2.0;
      BLD   103;
      AN    I     11.5;
      =     L      2.1;
      BLD   103;
      A     M     20.1;
      =     L      2.2;
      BLD   103;
      CALL FC   182 (
           IN0                      := L      2.0,
           IN1                      := L      2.1,
           IN2                      := L      2.2,
           OUT3                     := M    187.0,
           OUT4                     := M    187.1,
           OUT5                     := M    187.2,
           OUT6                     := DB10.DBW  320,
           IO7                      := DB182.DBW   30);
      NOP   0;
NETWORK
TITLE =

      A     M     21.0;
      =     L      2.0;
      BLD   103;
      AN    I     12.0;
      =     L      2.1;
      BLD   103;
      A     M     20.1;
      =     L      2.2;
      BLD   103;
      CALL FC   182 (
           IN0                      := L      2.0,
           IN1                      := L      2.1,
           IN2                      := L      2.2,
           OUT3                     := M    188.0,
           OUT4                     := M    188.1,
           OUT5                     := M    188.2,
           OUT6                     := DB10.DBW  322,
           IO7                      := DB182.DBW   32);
      NOP   0;
NETWORK
TITLE =

      A     M     21.0;
      =     L      2.0;
      BLD   103;
      AN    I     12.1;
      =     L      2.1;
      BLD   103;
      A     M     20.1;
      =     L      2.2;
      BLD   103;
      CALL FC   182 (
           IN0                      := L      2.0,
           IN1                      := L      2.1,
           IN2                      := L      2.2,
           OUT3                     := M    189.0,
           OUT4                     := M    189.1,
           OUT5                     := M    189.2,
           OUT6                     := DB10.DBW  324,
           IO7                      := DB182.DBW   34);
      NOP   0;
NETWORK
TITLE =

      A     M     21.0;
      =     L      2.0;
      BLD   103;
      A     I     12.2;
      =     L      2.1;
      BLD   103;
      A     M     20.1;
      =     L      2.2;
      BLD   103;
      CALL FC   182 (
           IN0                      := L      2.0,
           IN1                      := L      2.1,
           IN2                      := L      2.2,
           OUT3                     := M    190.0,
           OUT4                     := M    190.1,
           OUT5                     := M    190.2,
           OUT6                     := DB10.DBW  326,
           IO7                      := DB182.DBW   36);
      NOP   0;
NETWORK
TITLE =
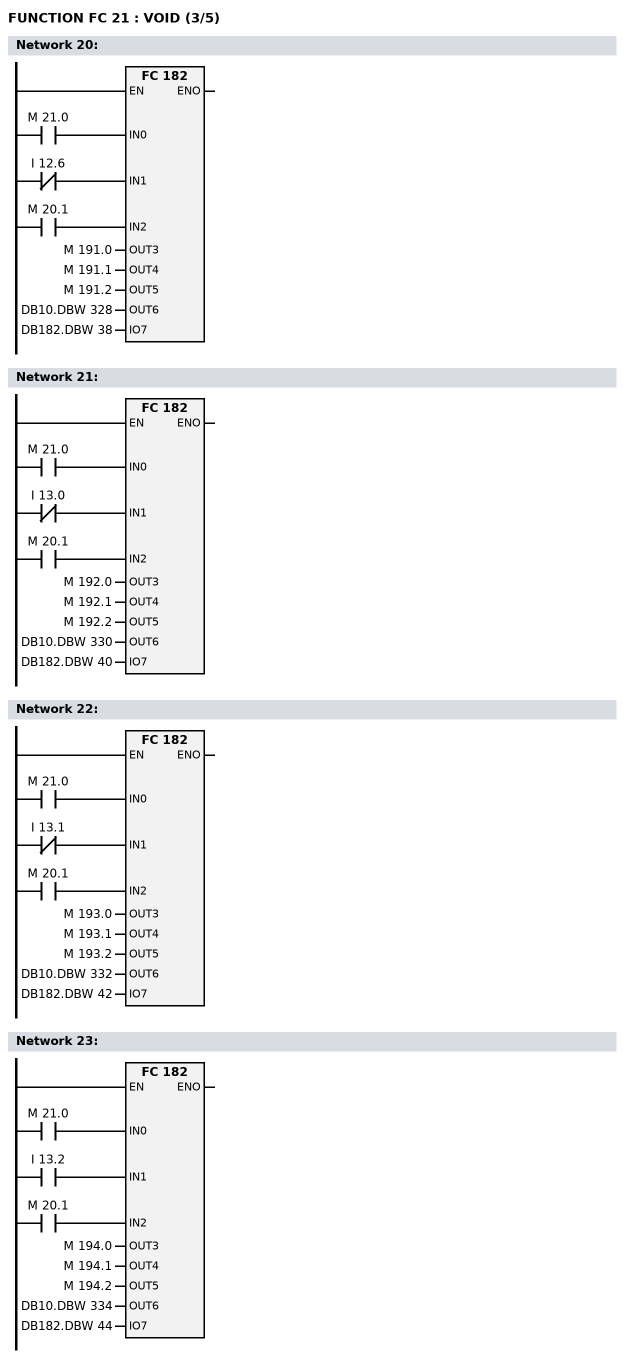

      A     M     21.0;
      =     L      2.0;
      BLD   103;
      AN    I     12.6;
      =     L      2.1;
      BLD   103;
      A     M     20.1;
      =     L      2.2;
      BLD   103;
      CALL FC   182 (
           IN0                      := L      2.0,
           IN1                      := L      2.1,
           IN2                      := L      2.2,
           OUT3                     := M    191.0,
           OUT4                     := M    191.1,
           OUT5                     := M    191.2,
           OUT6                     := DB10.DBW  328,
           IO7                      := DB182.DBW   38);
      NOP   0;
NETWORK
TITLE =

      A     M     21.0;
      =     L      2.0;
      BLD   103;
      AN    I     13.0;
      =     L      2.1;
      BLD   103;
      A     M     20.1;
      =     L      2.2;
      BLD   103;
      CALL FC   182 (
           IN0                      := L      2.0,
           IN1                      := L      2.1,
           IN2                      := L      2.2,
           OUT3                     := M    192.0,
           OUT4                     := M    192.1,
           OUT5                     := M    192.2,
           OUT6                     := DB10.DBW  330,
           IO7                      := DB182.DBW   40);
      NOP   0;
NETWORK
TITLE =

      A     M     21.0;
      =     L      2.0;
      BLD   103;
      AN    I     13.1;
      =     L      2.1;
      BLD   103;
      A     M     20.1;
      =     L      2.2;
      BLD   103;
      CALL FC   182 (
           IN0                      := L      2.0,
           IN1                      := L      2.1,
           IN2                      := L      2.2,
           OUT3                     := M    193.0,
           OUT4                     := M    193.1,
           OUT5                     := M    193.2,
           OUT6                     := DB10.DBW  332,
           IO7                      := DB182.DBW   42);
      NOP   0;
NETWORK
TITLE =

      A     M     21.0;
      =     L      2.0;
      BLD   103;
      A     I     13.2;
      =     L      2.1;
      BLD   103;
      A     M     20.1;
      =     L      2.2;
      BLD   103;
      CALL FC   182 (
           IN0                      := L      2.0,
           IN1                      := L      2.1,
           IN2                      := L      2.2,
           OUT3                     := M    194.0,
           OUT4                     := M    194.1,
           OUT5                     := M    194.2,
           OUT6                     := DB10.DBW  334,
           IO7                      := DB182.DBW   44);
      NOP   0;
NETWORK
TITLE =
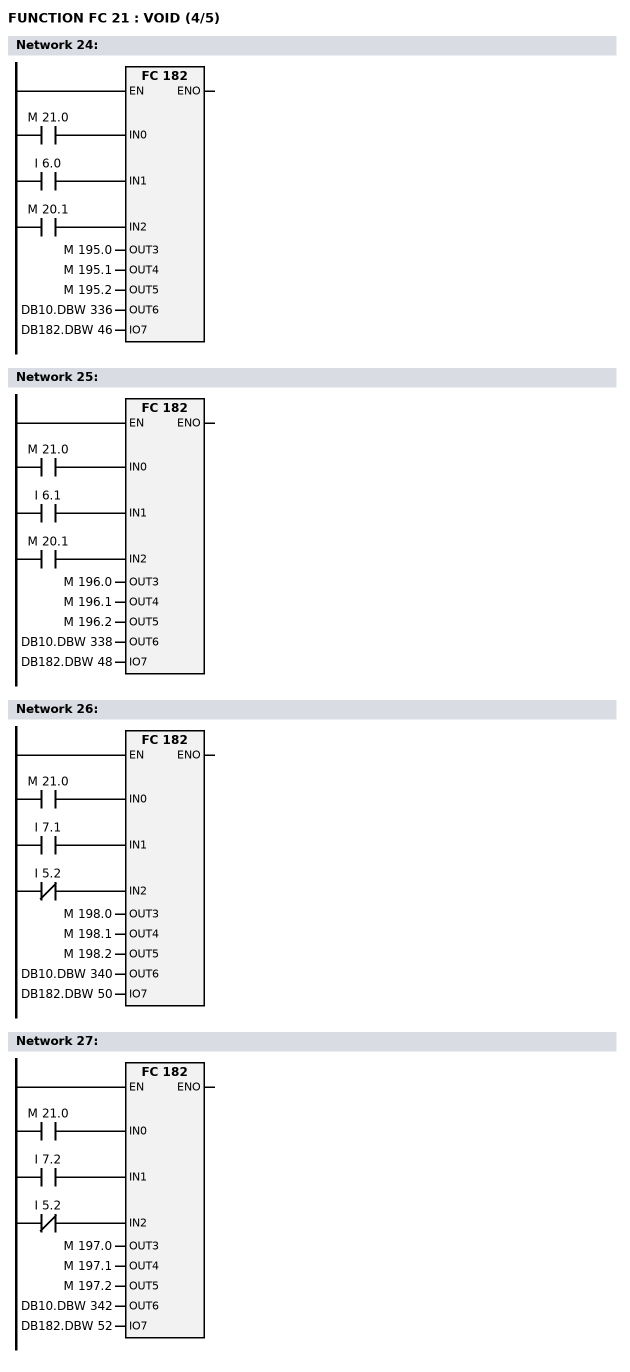

      A     M     21.0;
      =     L      2.0;
      BLD   103;
      A     I      6.0;
      =     L      2.1;
      BLD   103;
      A     M     20.1;
      =     L      2.2;
      BLD   103;
      CALL FC   182 (
           IN0                      := L      2.0,
           IN1                      := L      2.1,
           IN2                      := L      2.2,
           OUT3                     := M    195.0,
           OUT4                     := M    195.1,
           OUT5                     := M    195.2,
           OUT6                     := DB10.DBW  336,
           IO7                      := DB182.DBW   46);
      NOP   0;
NETWORK
TITLE =

      A     M     21.0;
      =     L      2.0;
      BLD   103;
      A     I      6.1;
      =     L      2.1;
      BLD   103;
      A     M     20.1;
      =     L      2.2;
      BLD   103;
      CALL FC   182 (
           IN0                      := L      2.0,
           IN1                      := L      2.1,
           IN2                      := L      2.2,
           OUT3                     := M    196.0,
           OUT4                     := M    196.1,
           OUT5                     := M    196.2,
           OUT6                     := DB10.DBW  338,
           IO7                      := DB182.DBW   48);
      NOP   0;
NETWORK
TITLE =

      A     M     21.0;
      =     L      2.0;
      BLD   103;
      A     I      7.1;
      =     L      2.1;
      BLD   103;
      AN    I      5.2;
      =     L      2.2;
      BLD   103;
      CALL FC   182 (
           IN0                      := L      2.0,
           IN1                      := L      2.1,
           IN2                      := L      2.2,
           OUT3                     := M    198.0,
           OUT4                     := M    198.1,
           OUT5                     := M    198.2,
           OUT6                     := DB10.DBW  340,
           IO7                      := DB182.DBW   50);
      NOP   0;
NETWORK
TITLE =

      A     M     21.0;
      =     L      2.0;
      BLD   103;
      A     I      7.2;
      =     L      2.1;
      BLD   103;
      AN    I      5.2;
      =     L      2.2;
      BLD   103;
      CALL FC   182 (
           IN0                      := L      2.0,
           IN1                      := L      2.1,
           IN2                      := L      2.2,
           OUT3                     := M    197.0,
           OUT4                     := M    197.1,
           OUT5                     := M    197.2,
           OUT6                     := DB10.DBW  342,
           IO7                      := DB182.DBW   52);
      NOP   0;
NETWORK
TITLE =
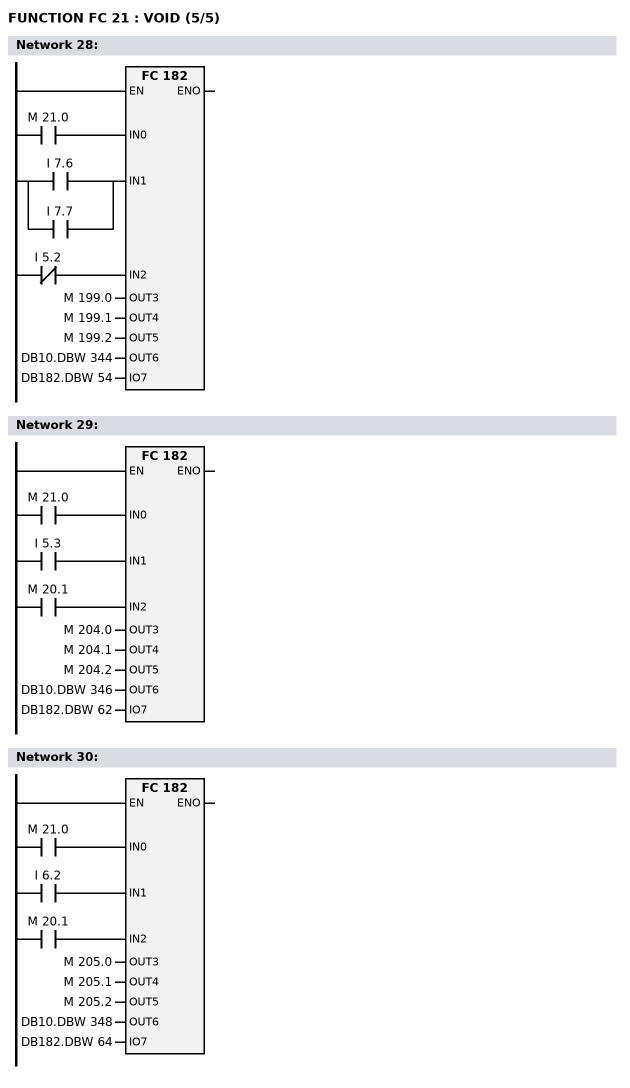

      A     M     21.0;
      =     L      2.0;
      BLD   103;
      A(    ;
      O     I      7.6;
      O     I      7.7;
      )     ;
      =     L      2.1;
      BLD   103;
      AN    I      5.2;
      =     L      2.2;
      BLD   103;
      CALL FC   182 (
           IN0                      := L      2.0,
           IN1                      := L      2.1,
           IN2                      := L      2.2,
           OUT3                     := M    199.0,
           OUT4                     := M    199.1,
           OUT5                     := M    199.2,
           OUT6                     := DB10.DBW  344,
           IO7                      := DB182.DBW   54);
      NOP   0;
NETWORK
TITLE =

      A     M     21.0;
      =     L      2.0;
      BLD   103;
      A     I      5.3;
      =     L      2.1;
      BLD   103;
      A     M     20.1;
      =     L      2.2;
      BLD   103;
      CALL FC   182 (
           IN0                      := L      2.0,
           IN1                      := L      2.1,
           IN2                      := L      2.2,
           OUT3                     := M    204.0,
           OUT4                     := M    204.1,
           OUT5                     := M    204.2,
           OUT6                     := DB10.DBW  346,
           IO7                      := DB182.DBW   62);
      NOP   0;
NETWORK
TITLE =

      A     M     21.0;
      =     L      2.0;
      BLD   103;
      A     I      6.2;
      =     L      2.1;
      BLD   103;
      A     M     20.1;
      =     L      2.2;
      BLD   103;
      CALL FC   182 (
           IN0                      := L      2.0,
           IN1                      := L      2.1,
           IN2                      := L      2.2,
           OUT3                     := M    205.0,
           OUT4                     := M    205.1,
           OUT5                     := M    205.2,
           OUT6                     := DB10.DBW  348,
           IO7                      := DB182.DBW   64);
      NOP   0;
END_FUNCTION

FUNCTION FC 3 : VOID
TITLE =
AUTHOR : Xaadem <yalanci63@yahoo.com>
FAMILY : Alarm
NAME : Alarm
VERSION : 0.1

BEGIN
NETWORK
TITLE =
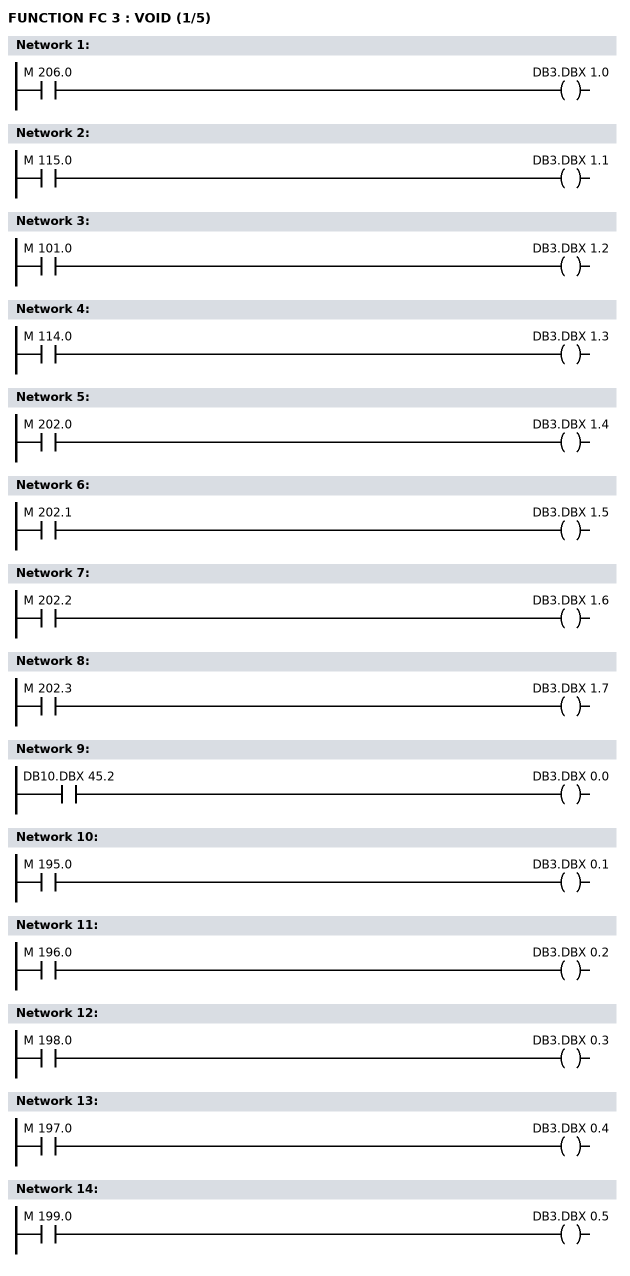

      A     M    206.0;
      =     DB3.DBX    1.0;
NETWORK
TITLE =

      A     M    115.0;
      =     DB3.DBX    1.1;
NETWORK
TITLE =

      A     M    101.0;
      =     DB3.DBX    1.2;
NETWORK
TITLE =

      A     M    114.0;
      =     DB3.DBX    1.3;
NETWORK
TITLE =

      A     M    202.0;
      =     DB3.DBX    1.4;
NETWORK
TITLE =

      A     M    202.1;
      =     DB3.DBX    1.5;
NETWORK
TITLE =

      A     M    202.2;
      =     DB3.DBX    1.6;
NETWORK
TITLE =

      A     M    202.3;
      =     DB3.DBX    1.7;
NETWORK
TITLE =

      A     DB10.DBX   45.2;
      =     DB3.DBX    0.0;
NETWORK
TITLE =

      A     M    195.0;
      =     DB3.DBX    0.1;
NETWORK
TITLE =

      A     M    196.0;
      =     DB3.DBX    0.2;
NETWORK
TITLE =

      A     M    198.0;
      =     DB3.DBX    0.3;
NETWORK
TITLE =

      A     M    197.0;
      =     DB3.DBX    0.4;
NETWORK
TITLE =

      A     M    199.0;
      =     DB3.DBX    0.5;
NETWORK
TITLE =
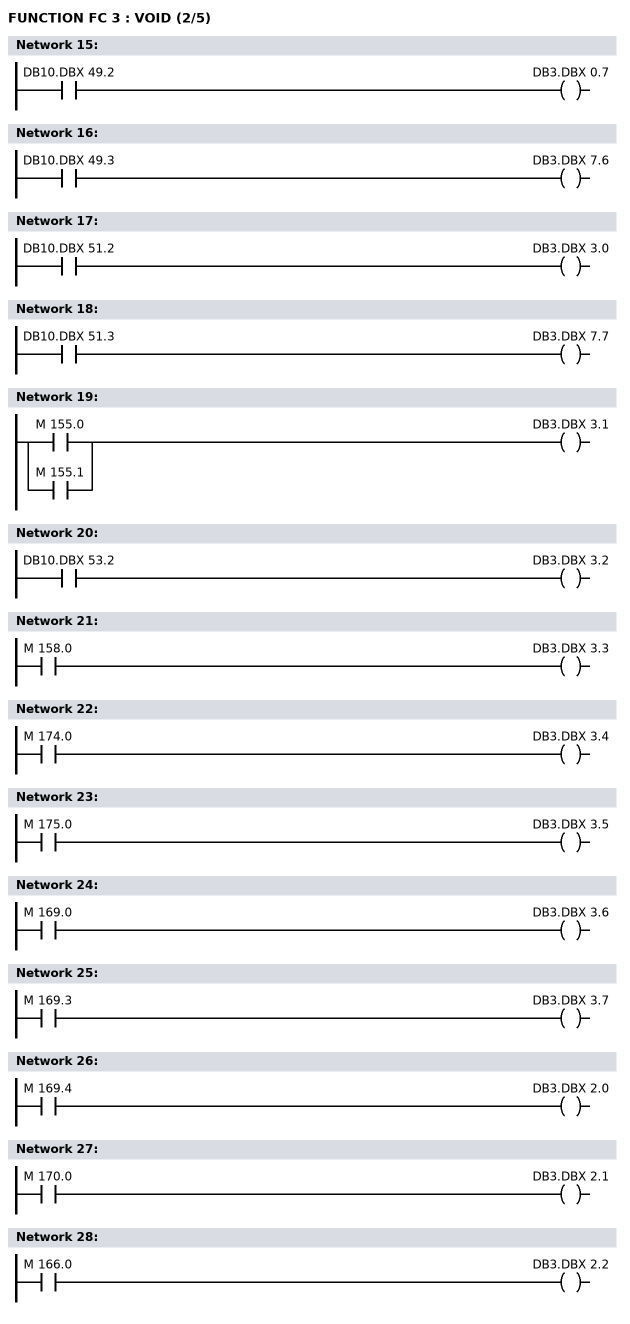

      A     DB10.DBX   49.2;
      =     DB3.DBX    0.7;
NETWORK
TITLE =

      A     DB10.DBX   49.3;
      =     DB3.DBX    7.6;
NETWORK
TITLE =

      A     DB10.DBX   51.2;
      =     DB3.DBX    3.0;
NETWORK
TITLE =

      A     DB10.DBX   51.3;
      =     DB3.DBX    7.7;
NETWORK
TITLE =

      O     M    155.0;
      O     M    155.1;
      =     DB3.DBX    3.1;
NETWORK
TITLE =

      A     DB10.DBX   53.2;
      =     DB3.DBX    3.2;
NETWORK
TITLE =

      A     M    158.0;
      =     DB3.DBX    3.3;
NETWORK
TITLE =

      A     M    174.0;
      =     DB3.DBX    3.4;
NETWORK
TITLE =

      A     M    175.0;
      =     DB3.DBX    3.5;
NETWORK
TITLE =

      A     M    169.0;
      =     DB3.DBX    3.6;
NETWORK
TITLE =

      A     M    169.3;
      =     DB3.DBX    3.7;
NETWORK
TITLE =

      A     M    169.4;
      =     DB3.DBX    2.0;
NETWORK
TITLE =

      A     M    170.0;
      =     DB3.DBX    2.1;
NETWORK
TITLE =

      A     M    166.0;
      =     DB3.DBX    2.2;
NETWORK
TITLE =
